FUNCTION_BLOCK Sensor_StateMonitor_View
  (* Version 0.1, 2005-12-15, Oscar Ljungkrantz, Chalmers *)
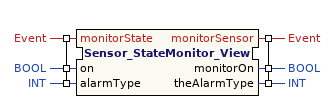
  EVENT_INPUT
    monitorState WITH on, alarmType;
  END_EVENT
  EVENT_OUTPUT
    monitorSensor WITH monitorOn, theAlarmType;
  END_EVENT
  VAR_INPUT
    on : BOOL;
    alarmType : INT;
  END_VAR
  VAR_OUTPUT
    monitorOn : BOOL;
    theAlarmType : INT;
  END_VAR
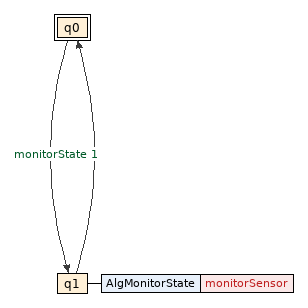
  EC_STATES
    q0;
    q1 : AlgMonitorState -> monitorSensor;
  END_STATES
  EC_TRANSITIONS
    q0 TO q1 := monitorState;
    q1 TO q0 := 1;
  END_TRANSITIONS
  ALGORITHM AlgMonitorState IN Java:
		monitorOn = on;
		theAlarmType = alarmType;
  END_ALGORITHM
END_FUNCTION_BLOCK
